// TIA Portal V18 export
// export: Created 2026-06-08T17:01:57.860434Z, ExportSetting WithDefaults, DisplayName Totally Integrated Automation Portal, DisplayVersion V18, DisplayName TIA Portal Openness, DisplayVersion V18, DisplayName TIA Portal Version Control Interface, DisplayVersion V18, DisplayName STEP 7 Professional, DisplayVersion V18, DisplayName STEP 7 Safety, DisplayVersion V18, DisplayName WinCC Professional, DisplayVersion V18
ORGANIZATION_BLOCK "Main"   // OB1, LAD, ProgramCycle
TITLE = "Main Program Sweep (Cycle)"
{ S7_Optimized_Access := 'TRUE' }
VERSION : 0.1
// stored: AutoNumber true, IsIECCheckEnabled false, SetENOAutomatically false
   VAR_INPUT
      Initial_Call : Bool;   // Initial call of this OB
      Remanence : Bool;   // =True, if remanent data are available
   END_VAR
BEGIN

REGION Network 1
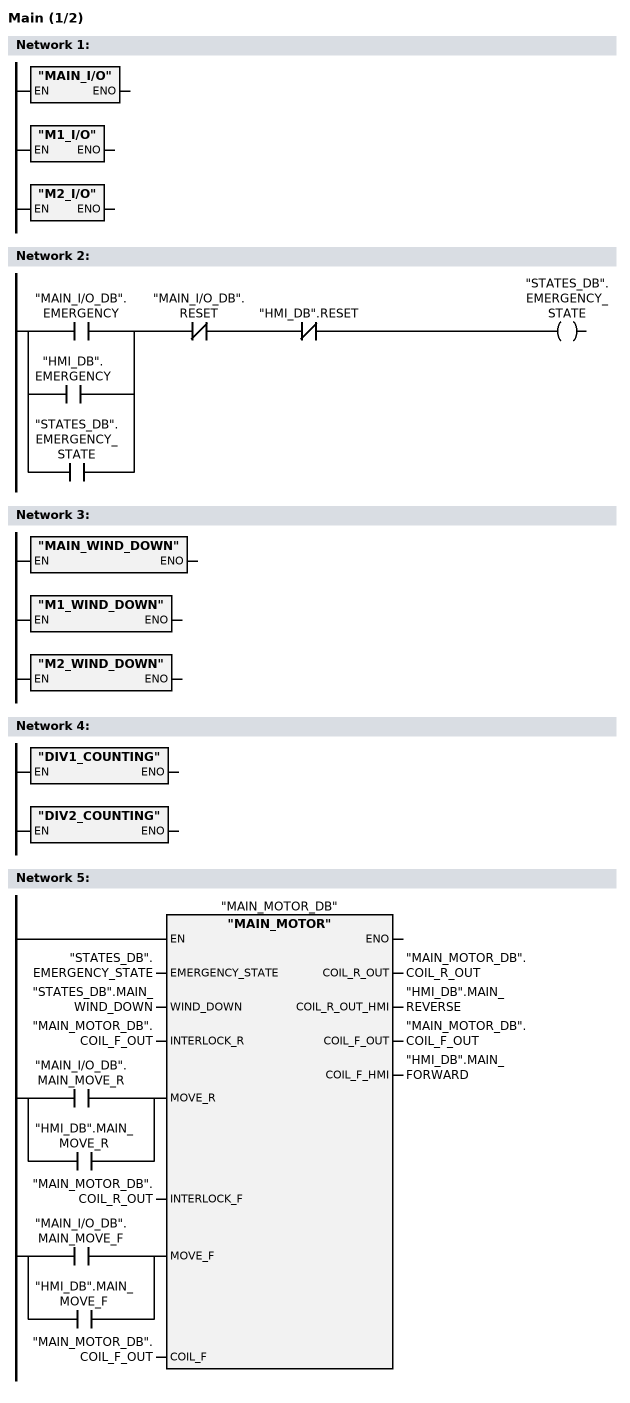
   RUNG wire#powerrail
      "MAIN_I/O"()
   END_RUNG
   RUNG wire#powerrail
      "M1_I/O"()
   END_RUNG
   RUNG wire#powerrail
      "M2_I/O"()
   END_RUNG
   // the same network as SCL:
   "MAIN_I/O"();
   "M1_I/O"();
   "M2_I/O"();
END_REGION

REGION Network 2
   RUNG wire#powerrail
      Contact( "MAIN_I/O_DB".EMERGENCY )
      wire#w1
      I_Contact( "MAIN_I/O_DB".RESET )
      I_Contact( "HMI_DB".RESET )
      Coil( "STATES_DB".EMERGENCY_STATE )
   END_RUNG
   RUNG wire#powerrail
      Contact( "HMI_DB".EMERGENCY )
   END_RUNG wire#w1
   RUNG wire#powerrail
      Contact( "STATES_DB".EMERGENCY_STATE )
   END_RUNG wire#w1
   // the same network as SCL:
   "STATES_DB".EMERGENCY_STATE := ("MAIN_I/O_DB".EMERGENCY OR "HMI_DB".EMERGENCY OR "STATES_DB".EMERGENCY_STATE) AND NOT "MAIN_I/O_DB".RESET AND NOT "HMI_DB".RESET;
END_REGION

REGION Network 3
   RUNG wire#powerrail
      "MAIN_WIND_DOWN"()
   END_RUNG
   RUNG wire#powerrail
      "M1_WIND_DOWN"()
   END_RUNG
   RUNG wire#powerrail
      "M2_WIND_DOWN"()
   END_RUNG
   // the same network as SCL:
   "MAIN_WIND_DOWN"();
   "M1_WIND_DOWN"();
   "M2_WIND_DOWN"();
END_REGION

REGION Network 4
   RUNG wire#powerrail
      "DIV1_COUNTING"()
   END_RUNG
   RUNG wire#powerrail
      "DIV2_COUNTING"()
   END_RUNG
   // the same network as SCL:
   "DIV1_COUNTING"();
   "DIV2_COUNTING"();
END_REGION

REGION Network 5
   RUNG wire#powerrail
      "MAIN_MOTOR_DB"(MOVE_R := wire#w1, MOVE_F := wire#w2, EMERGENCY_STATE := "STATES_DB".EMERGENCY_STATE, WIND_DOWN := "STATES_DB".MAIN_WIND_DOWN, INTERLOCK_R := "MAIN_MOTOR_DB".COIL_F_OUT, INTERLOCK_F := "MAIN_MOTOR_DB".COIL_R_OUT, COIL_F := "MAIN_MOTOR_DB".COIL_F_OUT, COIL_R_OUT => "MAIN_MOTOR_DB".COIL_R_OUT, COIL_R_OUT_HMI => "HMI_DB".MAIN_REVERSE, COIL_F_OUT => "MAIN_MOTOR_DB".COIL_F_OUT, COIL_F_HMI => "HMI_DB".MAIN_FORWARD)
   END_RUNG
   RUNG wire#powerrail
      Contact( "MAIN_I/O_DB".MAIN_MOVE_R )
   END_RUNG wire#w1
   RUNG wire#powerrail
      Contact( "HMI_DB".MAIN_MOVE_R )
   END_RUNG wire#w1
   RUNG wire#powerrail
      Contact( "MAIN_I/O_DB".MAIN_MOVE_F )
   END_RUNG wire#w2
   RUNG wire#powerrail
      Contact( "HMI_DB".MAIN_MOVE_F )
   END_RUNG wire#w2
   // the same network as SCL:
   "MAIN_MOTOR_DB"(EMERGENCY_STATE := "STATES_DB".EMERGENCY_STATE,   // "MAIN_MOTOR"
                   WIND_DOWN := "STATES_DB".MAIN_WIND_DOWN,
                   INTERLOCK_R := "MAIN_MOTOR_DB".COIL_F_OUT,
                   MOVE_R := "MAIN_I/O_DB".MAIN_MOVE_R OR "HMI_DB".MAIN_MOVE_R,
                   INTERLOCK_F := "MAIN_MOTOR_DB".COIL_R_OUT,
                   MOVE_F := "MAIN_I/O_DB".MAIN_MOVE_F OR "HMI_DB".MAIN_MOVE_F,
                   COIL_F := "MAIN_MOTOR_DB".COIL_F_OUT,
                   COIL_R_OUT => "MAIN_MOTOR_DB".COIL_R_OUT,
                   COIL_R_OUT_HMI => "HMI_DB".MAIN_REVERSE,
                   COIL_F_OUT => "MAIN_MOTOR_DB".COIL_F_OUT,
                   COIL_F_HMI => "HMI_DB".MAIN_FORWARD);
END_REGION

REGION Network 6
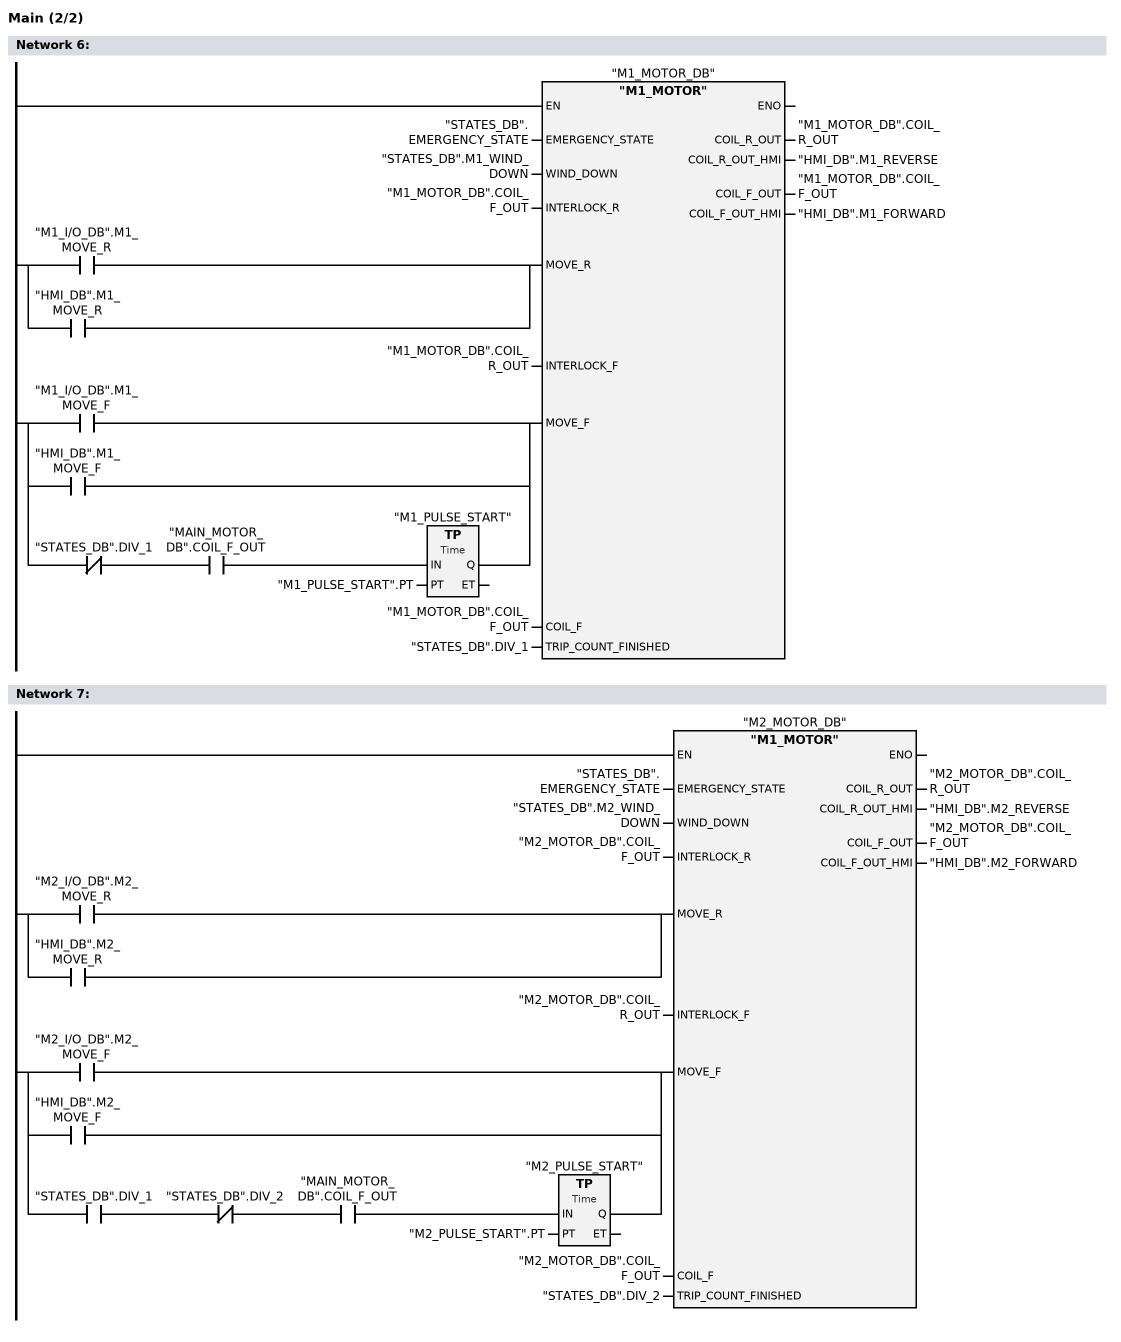
   RUNG wire#powerrail
      "M1_MOTOR_DB"(MOVE_R := wire#w1, MOVE_F := wire#w2, EMERGENCY_STATE := "STATES_DB".EMERGENCY_STATE, WIND_DOWN := "STATES_DB".M1_WIND_DOWN, INTERLOCK_R := "M1_MOTOR_DB".COIL_F_OUT, INTERLOCK_F := "M1_MOTOR_DB".COIL_R_OUT, COIL_F := "M1_MOTOR_DB".COIL_F_OUT, TRIP_COUNT_FINISHED := "STATES_DB".DIV_1, COIL_R_OUT => "M1_MOTOR_DB".COIL_R_OUT, COIL_R_OUT_HMI => "HMI_DB".M1_REVERSE, COIL_F_OUT => "M1_MOTOR_DB".COIL_F_OUT, COIL_F_OUT_HMI => "HMI_DB".M1_FORWARD)
   END_RUNG
   RUNG wire#powerrail
      Contact( "M1_I/O_DB".M1_MOVE_R )
   END_RUNG wire#w1
   RUNG wire#powerrail
      Contact( "HMI_DB".M1_MOVE_R )
   END_RUNG wire#w1
   RUNG wire#powerrail
      Contact( "M1_I/O_DB".M1_MOVE_F )
   END_RUNG wire#w2
   RUNG wire#powerrail
      Contact( "HMI_DB".M1_MOVE_F )
   END_RUNG wire#w2
   RUNG wire#powerrail
      I_Contact( "STATES_DB".DIV_1 )
      Contact( "MAIN_MOTOR_DB".COIL_F_OUT )
      { S7_Templates := "time_type := Time" } "M1_PULSE_START".TP(pt := "M1_PULSE_START".PT, et =>)
   END_RUNG wire#w2
   // the same network as SCL:
   "M1_PULSE_START".TP(IN := NOT "STATES_DB".DIV_1 AND "MAIN_MOTOR_DB".COIL_F_OUT, PT := "M1_PULSE_START".PT);
   "M1_MOTOR_DB"(EMERGENCY_STATE := "STATES_DB".EMERGENCY_STATE,   // "M1_MOTOR"
                 WIND_DOWN := "STATES_DB".M1_WIND_DOWN,
                 INTERLOCK_R := "M1_MOTOR_DB".COIL_F_OUT,
                 MOVE_R := "M1_I/O_DB".M1_MOVE_R OR "HMI_DB".M1_MOVE_R,
                 INTERLOCK_F := "M1_MOTOR_DB".COIL_R_OUT,
                 MOVE_F := "M1_I/O_DB".M1_MOVE_F OR "HMI_DB".M1_MOVE_F OR "M1_PULSE_START".Q,
                 COIL_F := "M1_MOTOR_DB".COIL_F_OUT,
                 TRIP_COUNT_FINISHED := "STATES_DB".DIV_1,
                 COIL_R_OUT => "M1_MOTOR_DB".COIL_R_OUT,
                 COIL_R_OUT_HMI => "HMI_DB".M1_REVERSE,
                 COIL_F_OUT => "M1_MOTOR_DB".COIL_F_OUT,
                 COIL_F_OUT_HMI => "HMI_DB".M1_FORWARD);
END_REGION

REGION Network 7
   RUNG wire#powerrail
      "M2_MOTOR_DB"(MOVE_R := wire#w1, MOVE_F := wire#w2, EMERGENCY_STATE := "STATES_DB".EMERGENCY_STATE, WIND_DOWN := "STATES_DB".M2_WIND_DOWN, INTERLOCK_R := "M2_MOTOR_DB".COIL_F_OUT, INTERLOCK_F := "M2_MOTOR_DB".COIL_R_OUT, COIL_F := "M2_MOTOR_DB".COIL_F_OUT, TRIP_COUNT_FINISHED := "STATES_DB".DIV_2, COIL_R_OUT => "M2_MOTOR_DB".COIL_R_OUT, COIL_R_OUT_HMI => "HMI_DB".M2_REVERSE, COIL_F_OUT => "M2_MOTOR_DB".COIL_F_OUT, COIL_F_OUT_HMI => "HMI_DB".M2_FORWARD)
   END_RUNG
   RUNG wire#powerrail
      Contact( "M2_I/O_DB".M2_MOVE_R )
   END_RUNG wire#w1
   RUNG wire#powerrail
      Contact( "HMI_DB".M2_MOVE_R )
   END_RUNG wire#w1
   RUNG wire#powerrail
      Contact( "M2_I/O_DB".M2_MOVE_F )
   END_RUNG wire#w2
   RUNG wire#powerrail
      Contact( "HMI_DB".M2_MOVE_F )
   END_RUNG wire#w2
   RUNG wire#powerrail
      Contact( "STATES_DB".DIV_1 )
      I_Contact( "STATES_DB".DIV_2 )
      Contact( "MAIN_MOTOR_DB".COIL_F_OUT )
      { S7_Templates := "time_type := Time" } "M2_PULSE_START".TP(pt := "M2_PULSE_START".PT, et =>)
   END_RUNG wire#w2
   // the same network as SCL:
   "M2_PULSE_START".TP(IN := "STATES_DB".DIV_1 AND NOT "STATES_DB".DIV_2 AND "MAIN_MOTOR_DB".COIL_F_OUT,
                       PT := "M2_PULSE_START".PT);
   "M2_MOTOR_DB"(EMERGENCY_STATE := "STATES_DB".EMERGENCY_STATE,   // "M1_MOTOR"
                 WIND_DOWN := "STATES_DB".M2_WIND_DOWN,
                 INTERLOCK_R := "M2_MOTOR_DB".COIL_F_OUT,
                 MOVE_R := "M2_I/O_DB".M2_MOVE_R OR "HMI_DB".M2_MOVE_R,
                 INTERLOCK_F := "M2_MOTOR_DB".COIL_R_OUT,
                 MOVE_F := "M2_I/O_DB".M2_MOVE_F OR "HMI_DB".M2_MOVE_F OR "M2_PULSE_START".Q,
                 COIL_F := "M2_MOTOR_DB".COIL_F_OUT,
                 TRIP_COUNT_FINISHED := "STATES_DB".DIV_2,
                 COIL_R_OUT => "M2_MOTOR_DB".COIL_R_OUT,
                 COIL_R_OUT_HMI => "HMI_DB".M2_REVERSE,
                 COIL_F_OUT => "M2_MOTOR_DB".COIL_F_OUT,
                 COIL_F_OUT_HMI => "HMI_DB".M2_FORWARD);
END_REGION
END_ORGANIZATION_BLOCK
